// TIA Portal V20 export
TYPE "LAxisCtrl_typePosRelative"
TITLE = LAxisCtrl_typePosRelative
// Support: tech.team.motioncontrol@siemens.com 
// Fax: +49 (0) 9131/98-1297
   STRUCT
      distance : LReal := 0.0;   // Distance for positioning process
      velocity : LReal := -1.0;   // Velocity setpoint for relative positioning (Value > 0.0: The specified value is used; Value = 0.0: Not permitted; Value < 0.0: Use of the default value configured in the technology object)
      acceleration : LReal := -1.0;   // Acceleration setpoint for relative positioning (Value > 0.0: The specified value is used; Value = 0.0: Not permitted; Value < 0.0: Use of the default value configured in the technology object)
      deceleration : LReal := -1.0;   // Deceleration setpoint for relative positioning (Value > 0.0: The specified value is used; Value = 0.0: Not permitted; Value < 0.0: Use of the default value configured in the technology object)
      jerk : LReal := -1.0;   // Jerk for relative positioning (Value > 0.0: Smooth velocity profile, the specified value is used; Value = 0.0: Trapezoid velocity profile; Value < 0.0: Use of the default value configured in the technology object)
      direction : DInt := 0;   // Motion direction of the axis (0: The sign of the distance parameter defines the direction; 1: Positive direction; 2: Negative direction)
   END_STRUCT;
END_TYPE
